INTERFACE PUBLIC HeldCommands EXTENDS RunningStateCommands

METHOD PUBLIC Unhold
END_METHOD

END_INTERFACE

(* stored: Version 1.1.0.1, ProductVersion 3.1.4026.18
   Itf HeldCommands: Id {39048063-0d8e-08f0-155a-0e9a16743f7e}
   Method Unhold: Id {b1afe03d-1a2c-0ac6-15ac-16a5319470a8} *)
